// SIMATIC S7-200 project (STEP 7-Micro/WIN), CPU 221 REL 01.10

ORGANIZATION_BLOCK PRINCIPAL:OB1
TITLE=COMENTARIOS DEL PROGRAMA
BEGIN
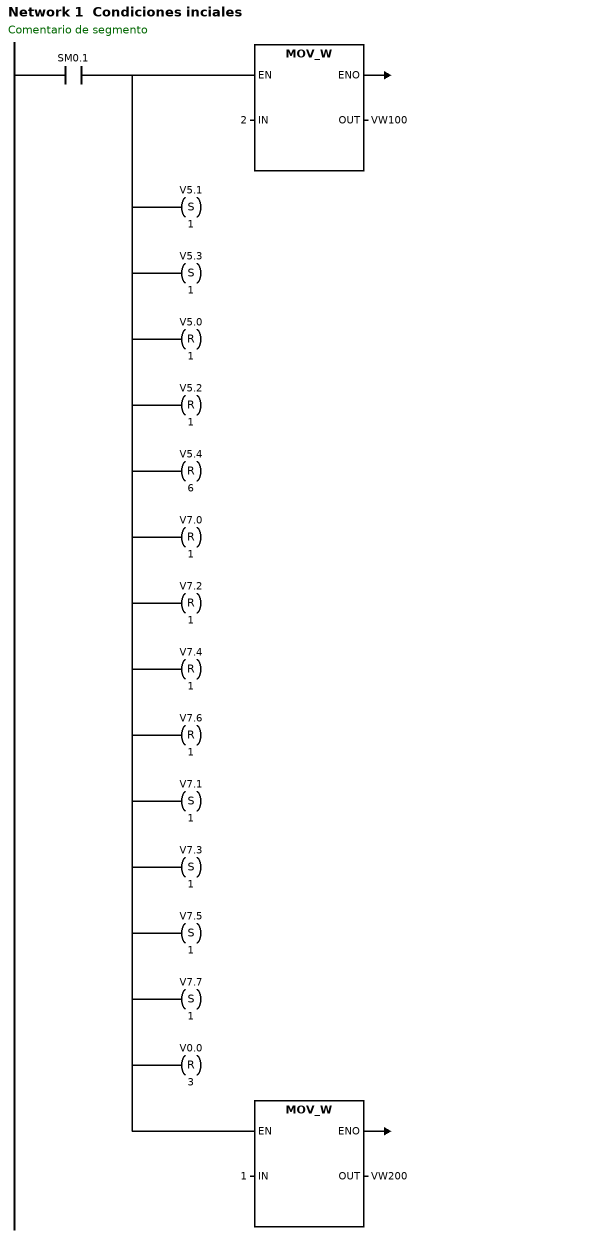
Network 1 // Condiciones inciales
// Comentario de segmento
LD     SM0.1
MOVW   2, VW100
S      V5.1, 1
S      V5.3, 1
R      V5.0, 1
R      V5.2, 1
R      V5.4, 6
R      V7.0, 1
R      V7.2, 1
R      V7.4, 1
R      V7.6, 1
S      V7.1, 1
S      V7.3, 1
S      V7.5, 1
S      V7.7, 1
R      V0.0, 3
MOVW   1, VW200
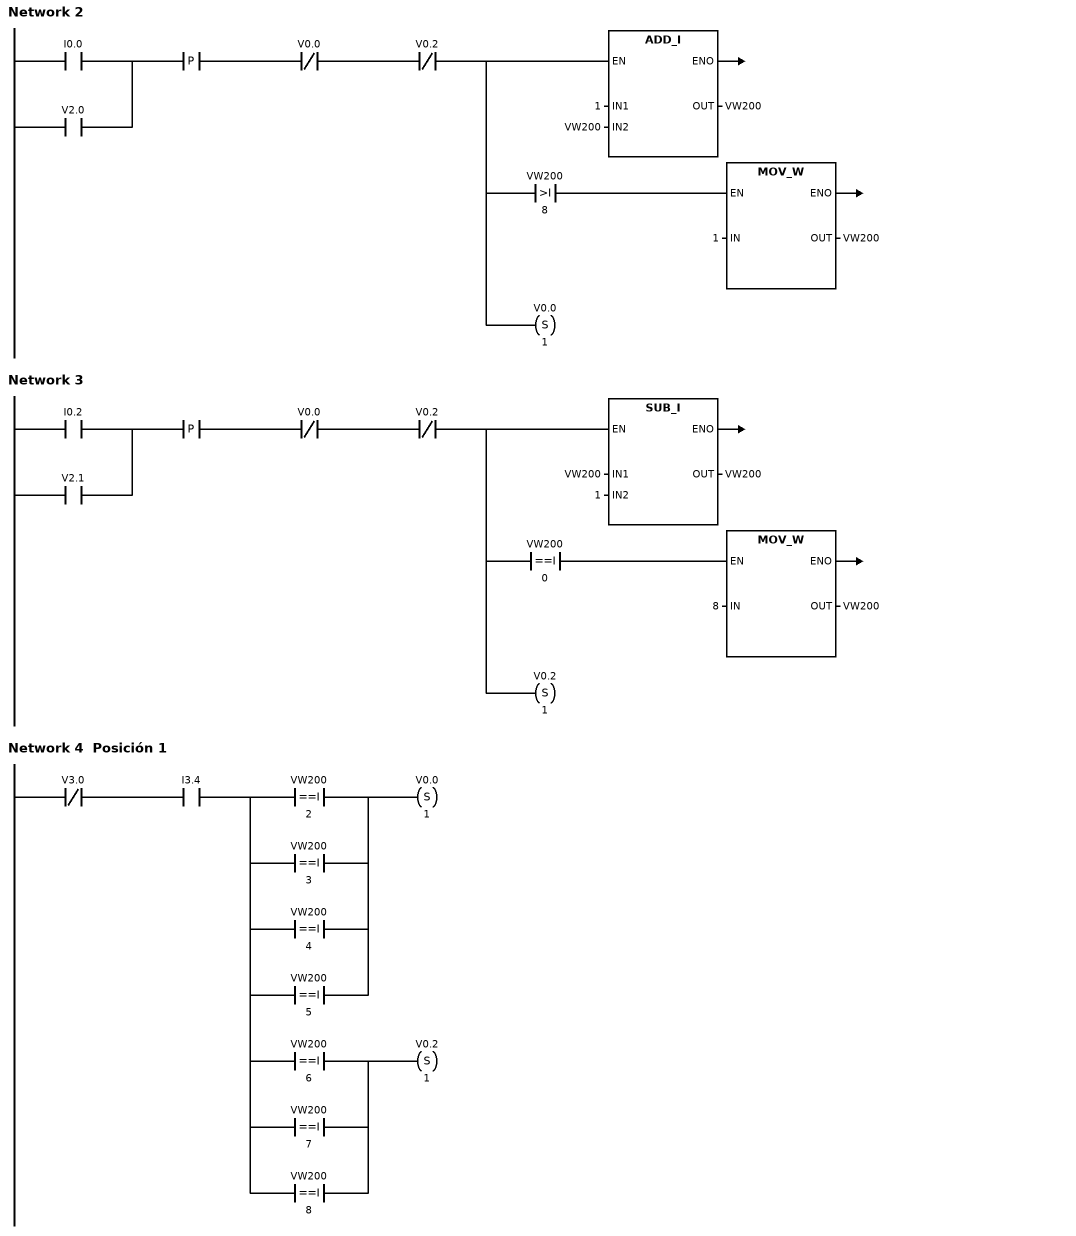
Network 2
LD     I0.0
O      V2.0
EU
AN     V0.0
AN     V0.2
LPS
+I     1, VW200
AW>    VW200, 8
MOVW   1, VW200
LPP
S      V0.0, 1
Network 3
LD     I0.2
O      V2.1
EU
AN     V0.0
AN     V0.2
LPS
-I     1, VW200
AW=    VW200, 0
MOVW   8, VW200
LPP
S      V0.2, 1
Network 4 // Posición 1
LDN    V3.0
A      I3.4
LPS
LDW=   VW200, 2
OW=    VW200, 3
OW=    VW200, 4
OW=    VW200, 5
ALD
S      V0.0, 1
LPP
LDW=   VW200, 6
OW=    VW200, 7
OW=    VW200, 8
ALD
S      V0.2, 1
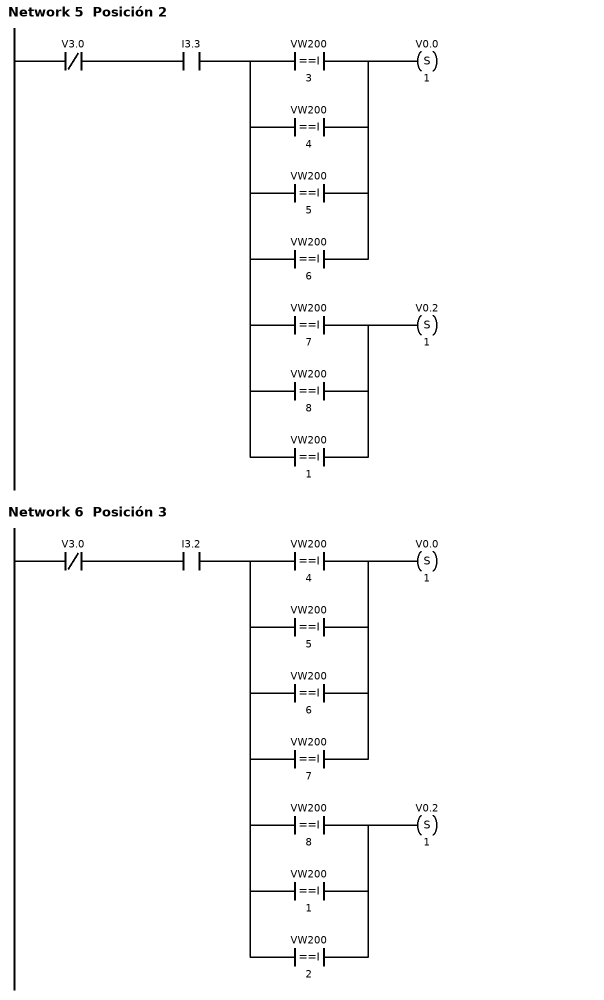
Network 5 // Posición 2
LDN    V3.0
A      I3.3
LPS
LDW=   VW200, 3
OW=    VW200, 4
OW=    VW200, 5
OW=    VW200, 6
ALD
S      V0.0, 1
LPP
LDW=   VW200, 7
OW=    VW200, 8
OW=    VW200, 1
ALD
S      V0.2, 1
Network 6 // Posición 3
LDN    V3.0
A      I3.2
LPS
LDW=   VW200, 4
OW=    VW200, 5
OW=    VW200, 6
OW=    VW200, 7
ALD
S      V0.0, 1
LPP
LDW=   VW200, 8
OW=    VW200, 1
OW=    VW200, 2
ALD
S      V0.2, 1
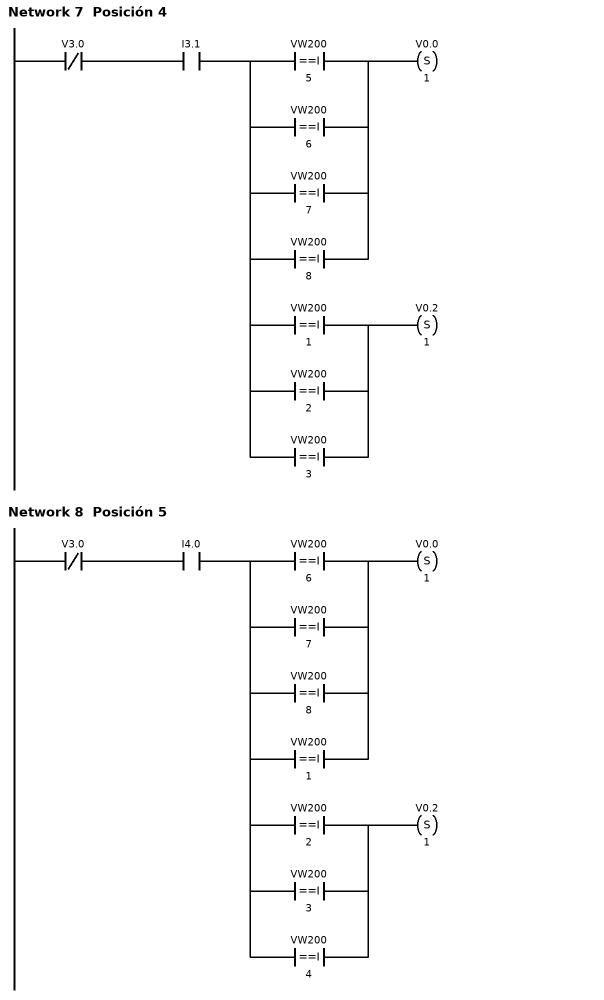
Network 7 // Posición 4
LDN    V3.0
A      I3.1
LPS
LDW=   VW200, 5
OW=    VW200, 6
OW=    VW200, 7
OW=    VW200, 8
ALD
S      V0.0, 1
LPP
LDW=   VW200, 1
OW=    VW200, 2
OW=    VW200, 3
ALD
S      V0.2, 1
Network 8 // Posición 5
LDN    V3.0
A      I4.0
LPS
LDW=   VW200, 6
OW=    VW200, 7
OW=    VW200, 8
OW=    VW200, 1
ALD
S      V0.0, 1
LPP
LDW=   VW200, 2
OW=    VW200, 3
OW=    VW200, 4
ALD
S      V0.2, 1
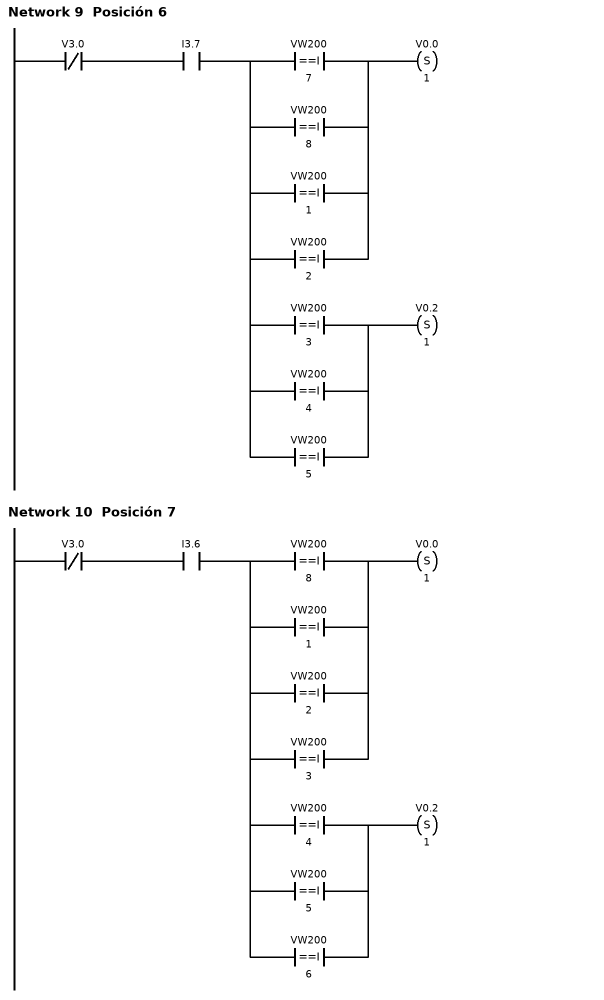
Network 9 // Posición 6
LDN    V3.0
A      I3.7
LPS
LDW=   VW200, 7
OW=    VW200, 8
OW=    VW200, 1
OW=    VW200, 2
ALD
S      V0.0, 1
LPP
LDW=   VW200, 3
OW=    VW200, 4
OW=    VW200, 5
ALD
S      V0.2, 1
Network 10 // Posición 7
LDN    V3.0
A      I3.6
LPS
LDW=   VW200, 8
OW=    VW200, 1
OW=    VW200, 2
OW=    VW200, 3
ALD
S      V0.0, 1
LPP
LDW=   VW200, 4
OW=    VW200, 5
OW=    VW200, 6
ALD
S      V0.2, 1
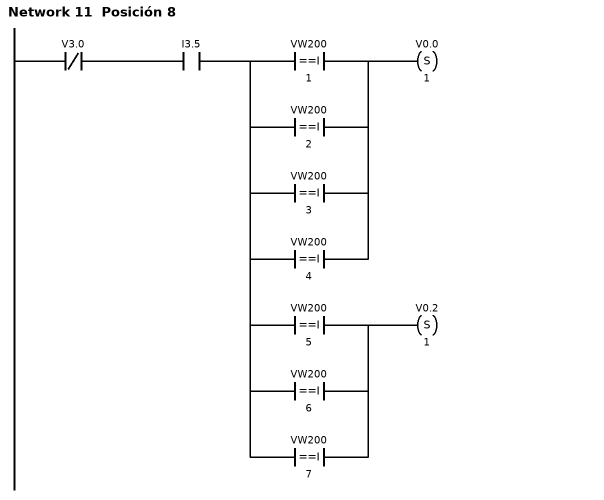
Network 11 // Posición 8
LDN    V3.0
A      I3.5
LPS
LDW=   VW200, 1
OW=    VW200, 2
OW=    VW200, 3
OW=    VW200, 4
ALD
S      V0.0, 1
LPP
LDW=   VW200, 5
OW=    VW200, 6
OW=    VW200, 7
ALD
S      V0.2, 1
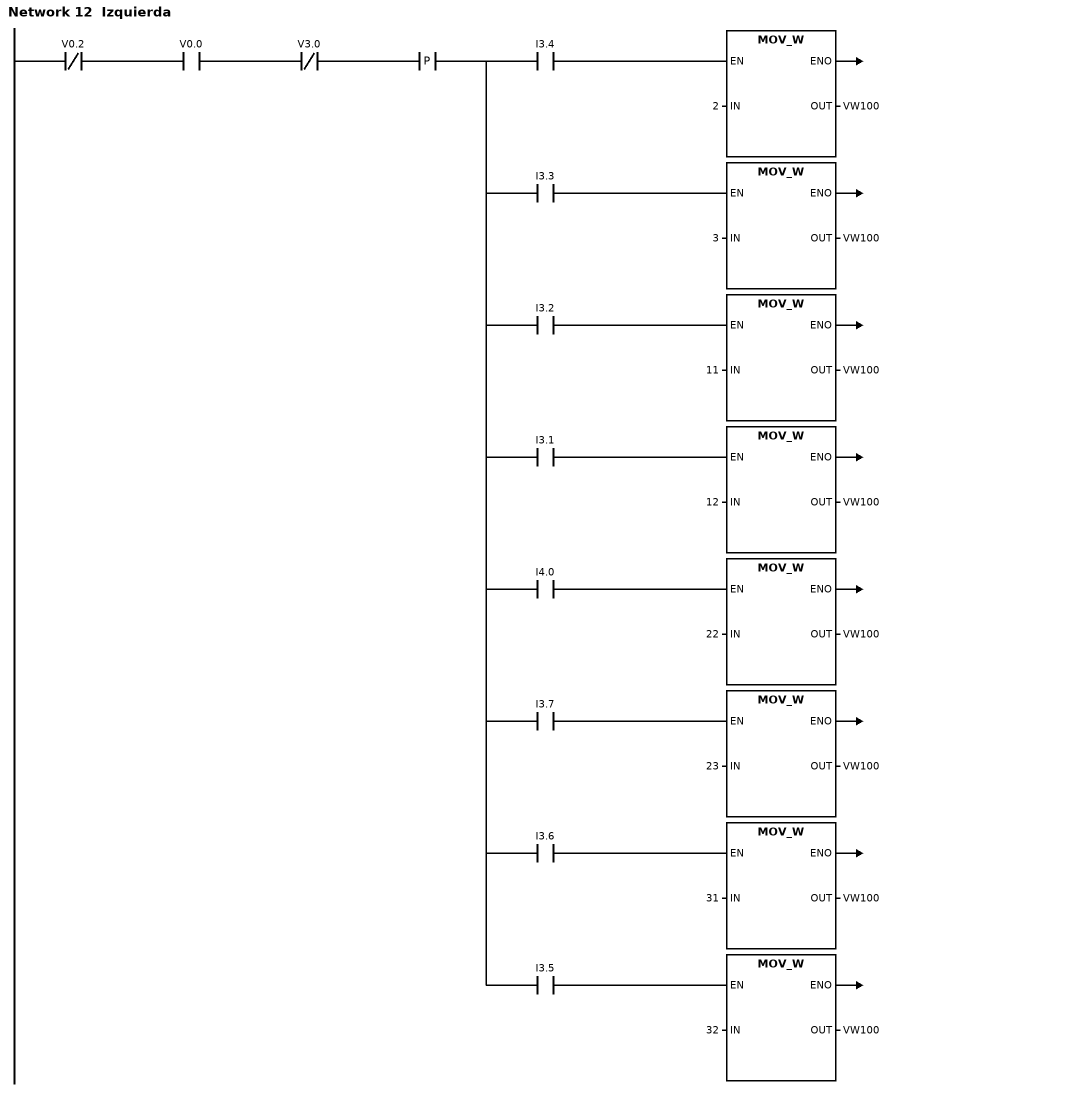
Network 12 // Izquierda
LDN    V0.2
A      V0.0
AN     V3.0
EU
LPS
A      I3.4
MOVW   2, VW100
LRD
A      I3.3
MOVW   3, VW100
LRD
A      I3.2
MOVW   11, VW100
LRD
A      I3.1
MOVW   12, VW100
LRD
A      I4.0
MOVW   22, VW100
LRD
A      I3.7
MOVW   23, VW100
LRD
A      I3.6
MOVW   31, VW100
LPP
A      I3.5
MOVW   32, VW100
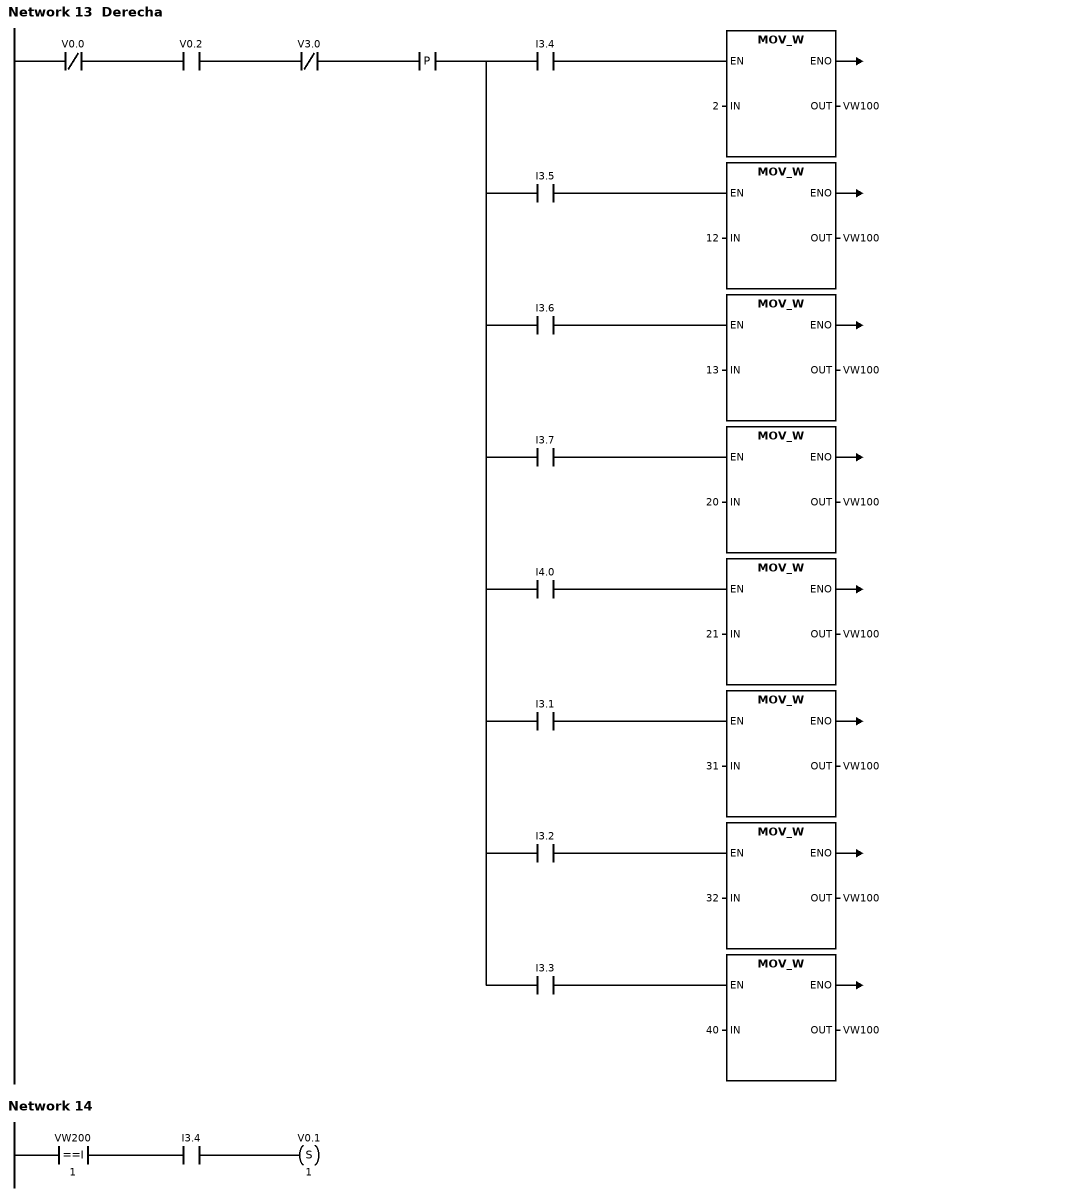
Network 13 // Derecha
LDN    V0.0
A      V0.2
AN     V3.0
EU
LPS
A      I3.4
MOVW   2, VW100
LRD
A      I3.5
MOVW   12, VW100
LRD
A      I3.6
MOVW   13, VW100
LRD
A      I3.7
MOVW   20, VW100
LRD
A      I4.0
MOVW   21, VW100
LRD
A      I3.1
MOVW   31, VW100
LRD
A      I3.2
MOVW   32, VW100
LPP
A      I3.3
MOVW   40, VW100
Network 14
LDW=   VW200, 1
A      I3.4
S      V0.1, 1
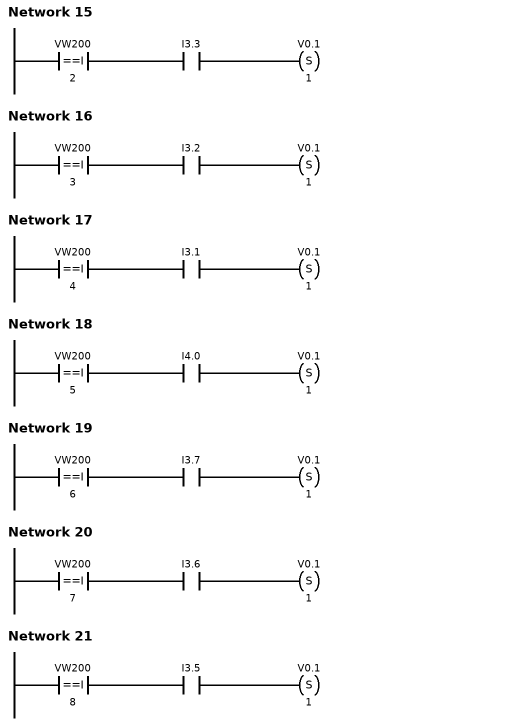
Network 15
LDW=   VW200, 2
A      I3.3
S      V0.1, 1
Network 16
LDW=   VW200, 3
A      I3.2
S      V0.1, 1
Network 17
LDW=   VW200, 4
A      I3.1
S      V0.1, 1
Network 18
LDW=   VW200, 5
A      I4.0
S      V0.1, 1
Network 19
LDW=   VW200, 6
A      I3.7
S      V0.1, 1
Network 20
LDW=   VW200, 7
A      I3.6
S      V0.1, 1
Network 21
LDW=   VW200, 8
A      I3.5
S      V0.1, 1
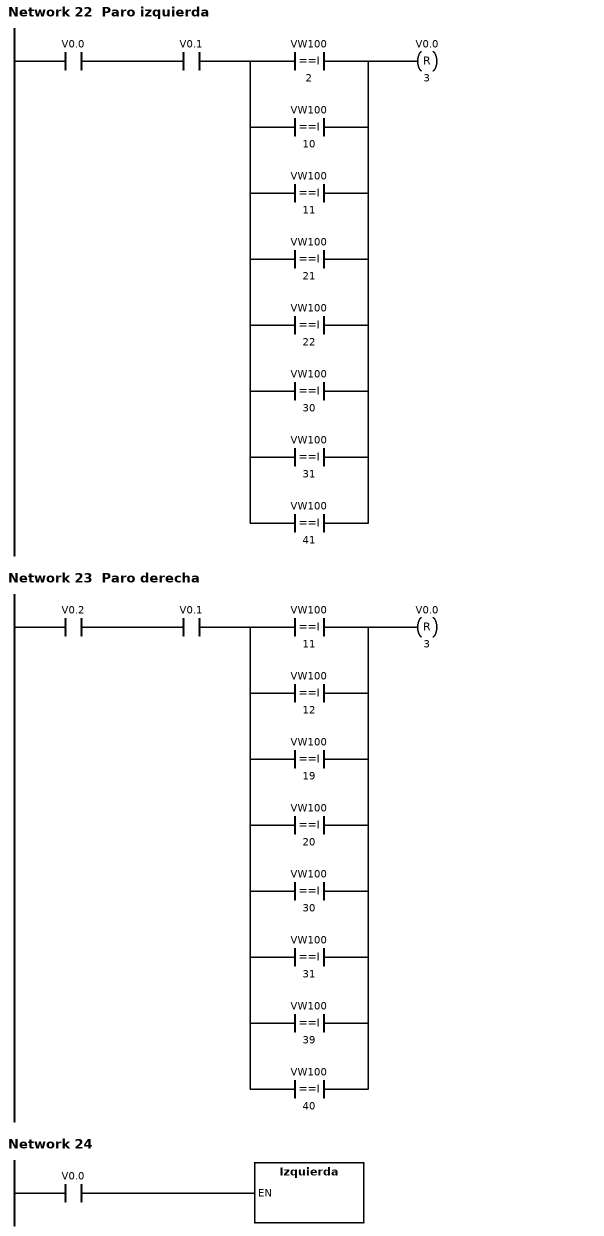
Network 22 // Paro izquierda
LD     V0.0
A      V0.1
LDW=   VW100, 2
OW=    VW100, 10
OW=    VW100, 11
OW=    VW100, 21
OW=    VW100, 22
OW=    VW100, 30
OW=    VW100, 31
OW=    VW100, 41
ALD
R      V0.0, 3
Network 23 // Paro derecha
LD     V0.2
A      V0.1
LDW=   VW100, 11
OW=    VW100, 12
OW=    VW100, 19
OW=    VW100, 20
OW=    VW100, 30
OW=    VW100, 31
OW=    VW100, 39
OW=    VW100, 40
ALD
R      V0.0, 3
Network 24
LD     V0.0
CALL   Izquierda:SBR0
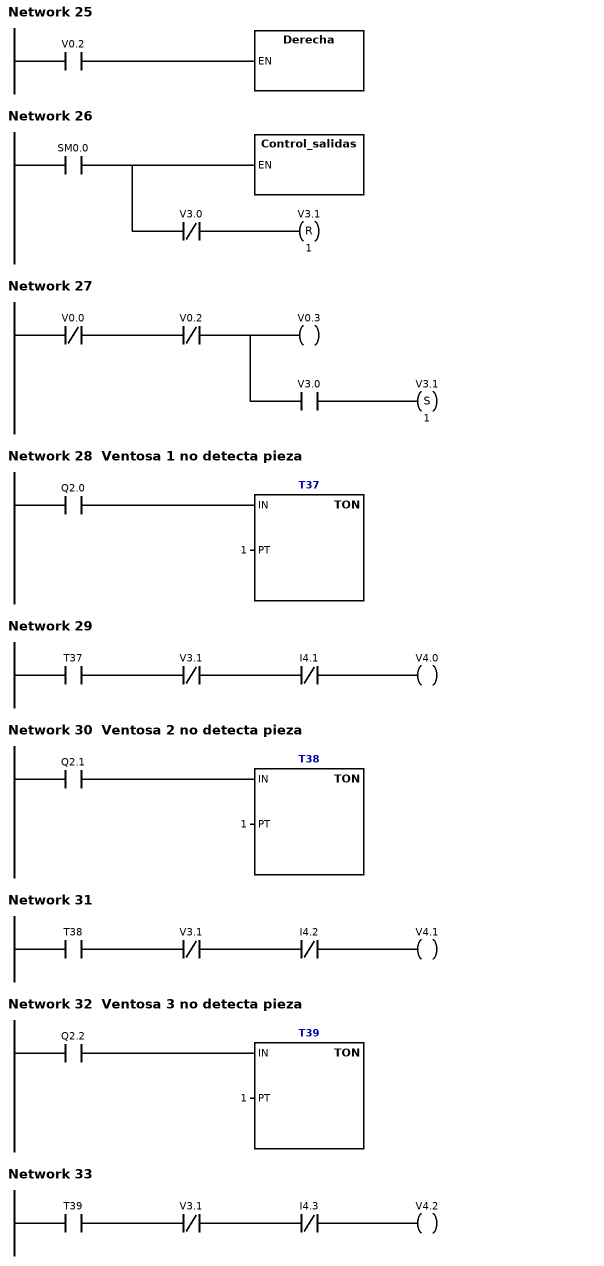
Network 25
LD     V0.2
CALL   Derecha:SBR1
Network 26
LD     SM0.0
CALL   Control_salidas:SBR2
AN     V3.0
R      V3.1, 1
Network 27
LDN    V0.0
AN     V0.2
=      V0.3
A      V3.0
S      V3.1, 1
Network 28 // Ventosa 1 no detecta pieza
LD     Q2.0
TON    T37, 1
Network 29
LD     T37
AN     V3.1
AN     I4.1
=      V4.0
Network 30 // Ventosa 2 no detecta pieza
LD     Q2.1
TON    T38, 1
Network 31
LD     T38
AN     V3.1
AN     I4.2
=      V4.1
Network 32 // Ventosa 3 no detecta pieza
LD     Q2.2
TON    T39, 1
Network 33
LD     T39
AN     V3.1
AN     I4.3
=      V4.2
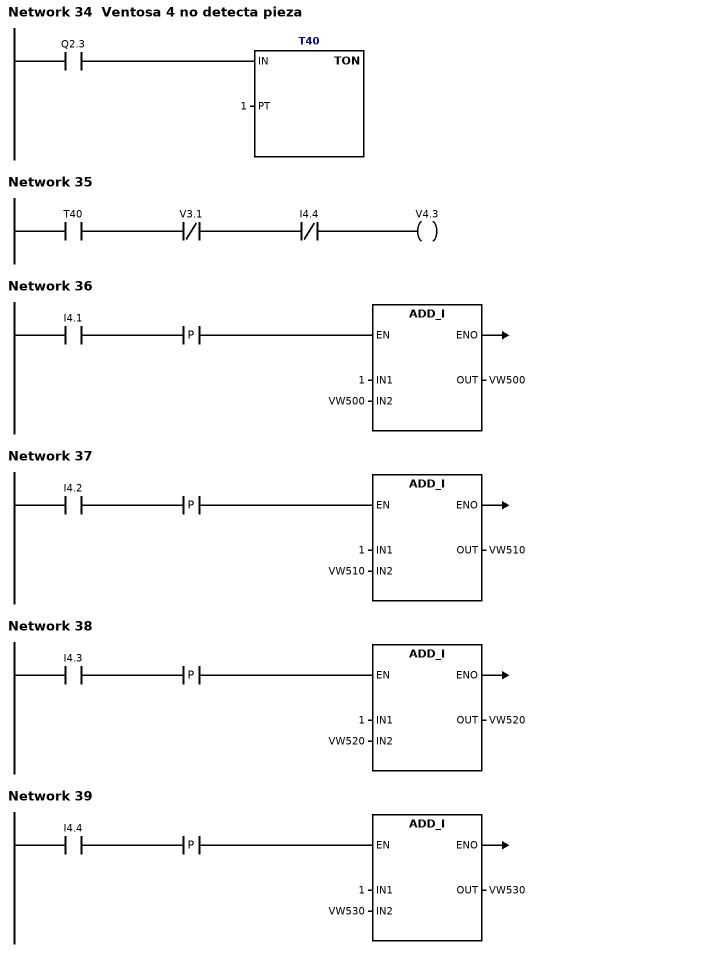
Network 34 // Ventosa 4 no detecta pieza
LD     Q2.3
TON    T40, 1
Network 35
LD     T40
AN     V3.1
AN     I4.4
=      V4.3
Network 36
LD     I4.1
EU
+I     1, VW500
Network 37
LD     I4.2
EU
+I     1, VW510
Network 38
LD     I4.3
EU
+I     1, VW520
Network 39
LD     I4.4
EU
+I     1, VW530
END_ORGANIZATION_BLOCK

SUBROUTINE_BLOCK Izquierda:SBR0
TITLE=COMENTARIOS DE LA SUBRUTINA
BEGIN
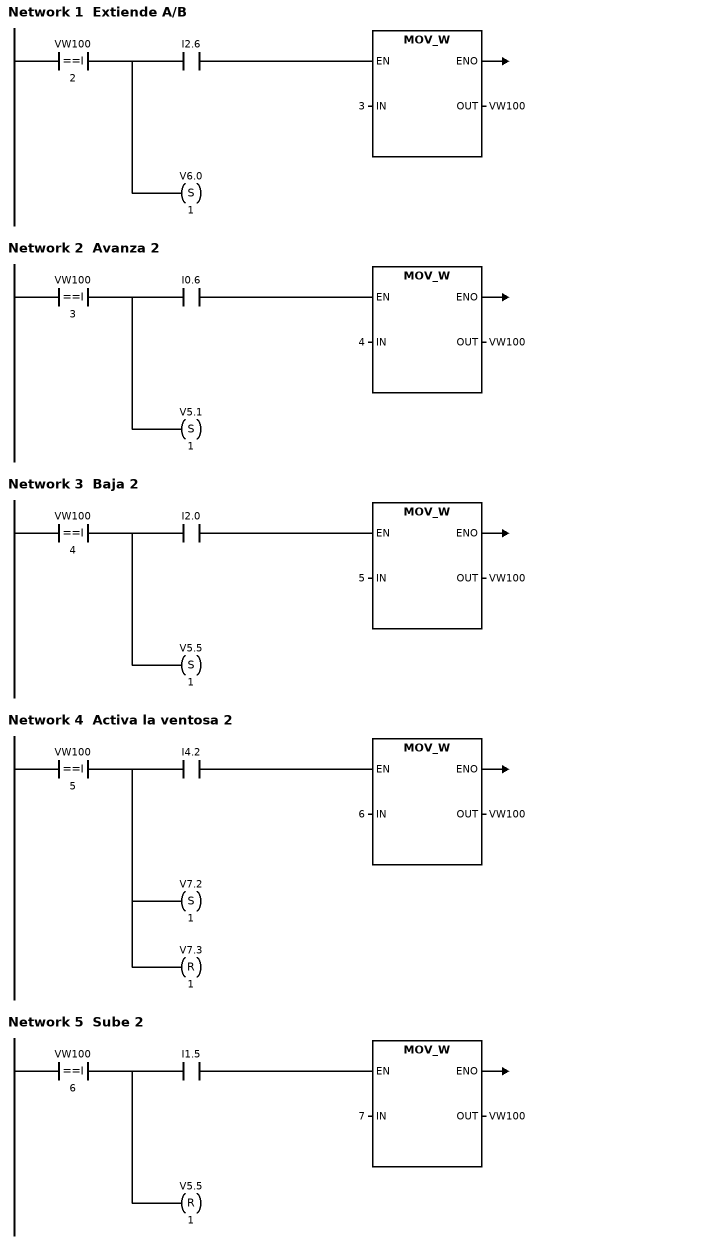
Network 1 // Extiende A/B
LDW=   VW100, 2
LPS
A      I2.6
MOVW   3, VW100
LPP
S      V6.0, 1
Network 2 // Avanza 2
LDW=   VW100, 3
LPS
A      I0.6
MOVW   4, VW100
LPP
S      V5.1, 1
Network 3 // Baja 2
LDW=   VW100, 4
LPS
A      I2.0
MOVW   5, VW100
LPP
S      V5.5, 1
Network 4 // Activa la ventosa 2
LDW=   VW100, 5
LPS
A      I4.2
MOVW   6, VW100
LRD
S      V7.2, 1
LPP
R      V7.3, 1
Network 5 // Sube 2
LDW=   VW100, 6
LPS
A      I1.5
MOVW   7, VW100
LPP
R      V5.5, 1
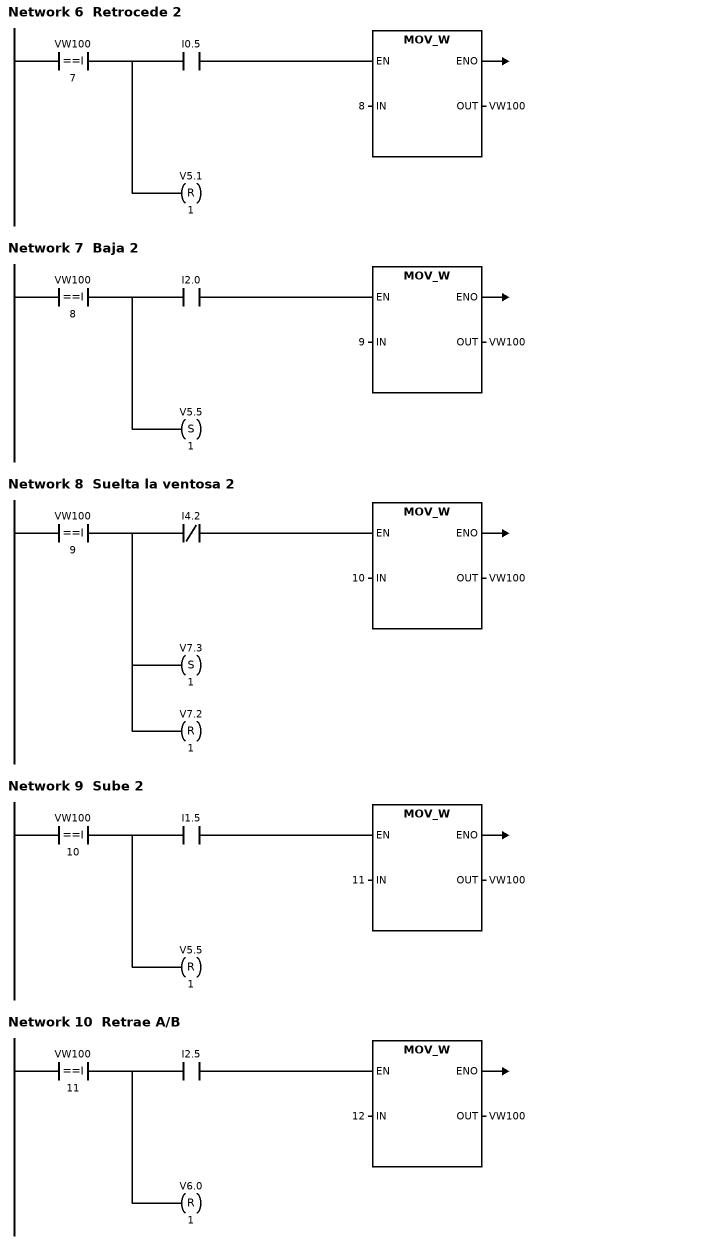
Network 6 // Retrocede 2
LDW=   VW100, 7
LPS
A      I0.5
MOVW   8, VW100
LPP
R      V5.1, 1
Network 7 // Baja 2
LDW=   VW100, 8
LPS
A      I2.0
MOVW   9, VW100
LPP
S      V5.5, 1
Network 8 // Suelta la ventosa 2
LDW=   VW100, 9
LPS
AN     I4.2
MOVW   10, VW100
LRD
S      V7.3, 1
LPP
R      V7.2, 1
Network 9 // Sube 2
LDW=   VW100, 10
LPS
A      I1.5
MOVW   11, VW100
LPP
R      V5.5, 1
Network 10 // Retrae A/B
LDW=   VW100, 11
LPS
A      I2.5
MOVW   12, VW100
LPP
R      V6.0, 1
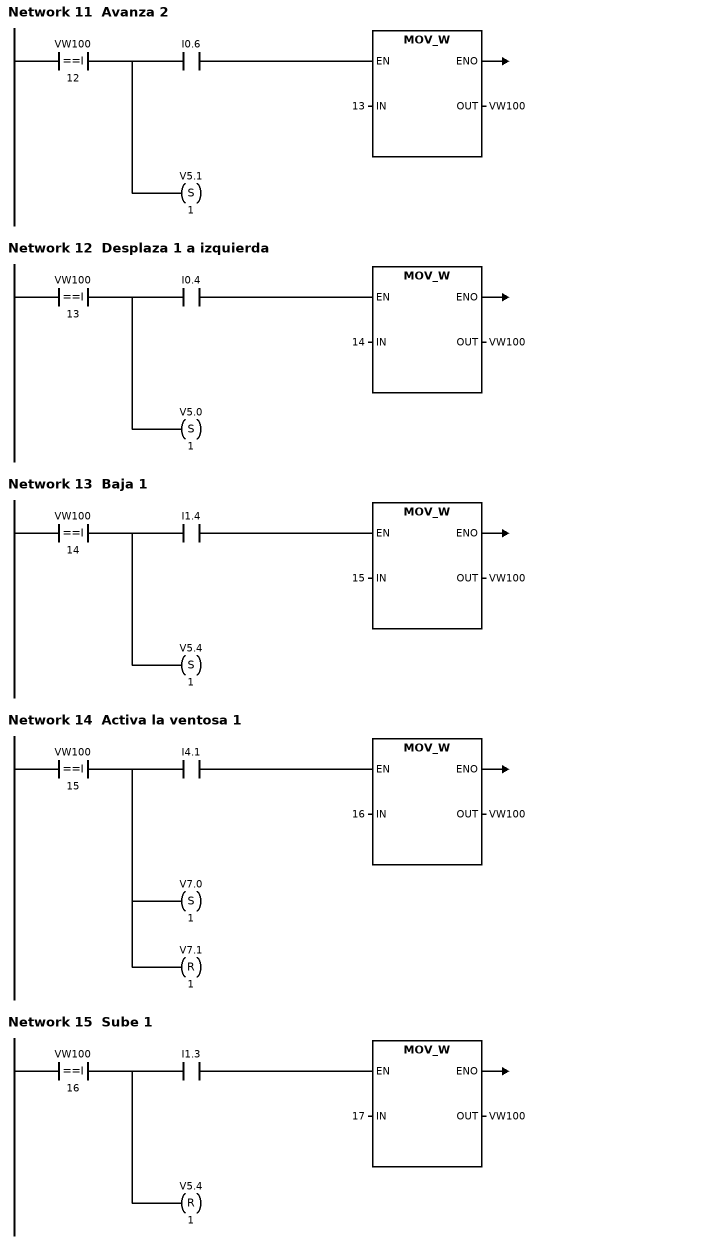
Network 11 // Avanza 2
LDW=   VW100, 12
LPS
A      I0.6
MOVW   13, VW100
LPP
S      V5.1, 1
Network 12 // Desplaza 1 a izquierda
LDW=   VW100, 13
LPS
A      I0.4
MOVW   14, VW100
LPP
S      V5.0, 1
Network 13 // Baja 1
LDW=   VW100, 14
LPS
A      I1.4
MOVW   15, VW100
LPP
S      V5.4, 1
Network 14 // Activa la ventosa 1
LDW=   VW100, 15
LPS
A      I4.1
MOVW   16, VW100
LRD
S      V7.0, 1
LPP
R      V7.1, 1
Network 15 // Sube 1
LDW=   VW100, 16
LPS
A      I1.3
MOVW   17, VW100
LPP
R      V5.4, 1
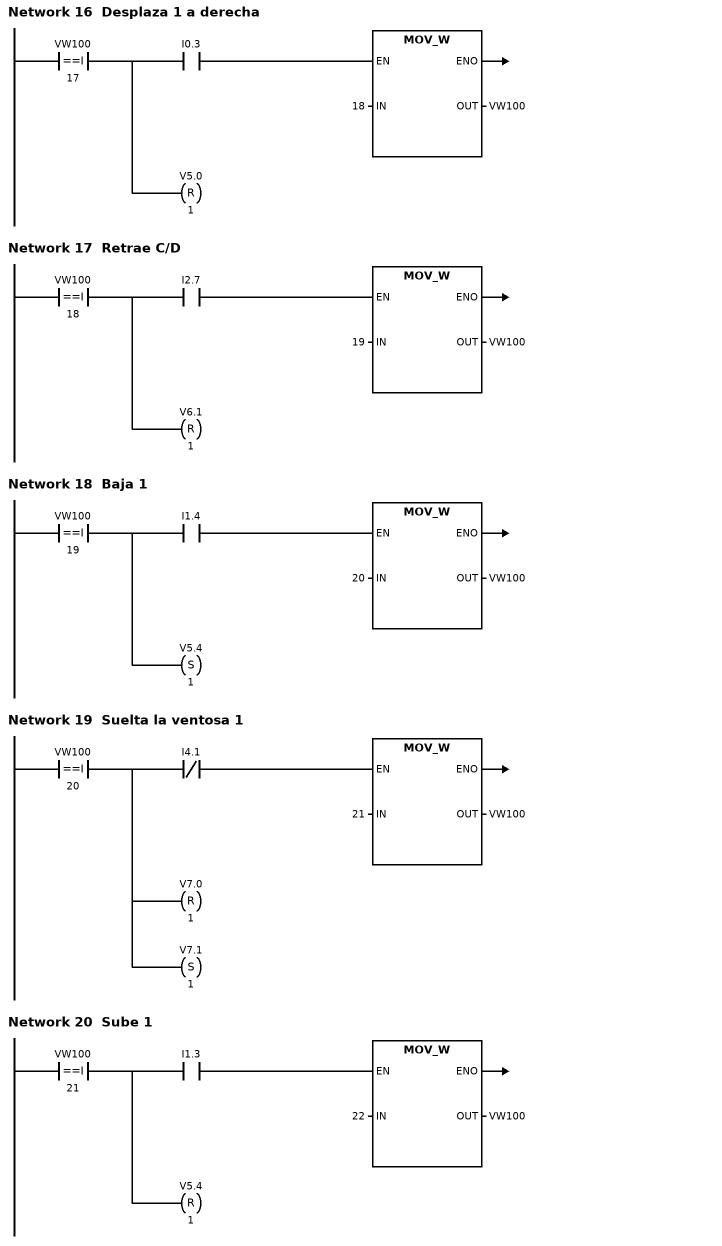
Network 16 // Desplaza 1 a derecha
LDW=   VW100, 17
LPS
A      I0.3
MOVW   18, VW100
LPP
R      V5.0, 1
Network 17 // Retrae C/D
LDW=   VW100, 18
LPS
A      I2.7
MOVW   19, VW100
LPP
R      V6.1, 1
Network 18 // Baja 1
LDW=   VW100, 19
LPS
A      I1.4
MOVW   20, VW100
LPP
S      V5.4, 1
Network 19 // Suelta la ventosa 1
LDW=   VW100, 20
LPS
AN     I4.1
MOVW   21, VW100
LRD
R      V7.0, 1
LPP
S      V7.1, 1
Network 20 // Sube 1
LDW=   VW100, 21
LPS
A      I1.3
MOVW   22, VW100
LPP
R      V5.4, 1
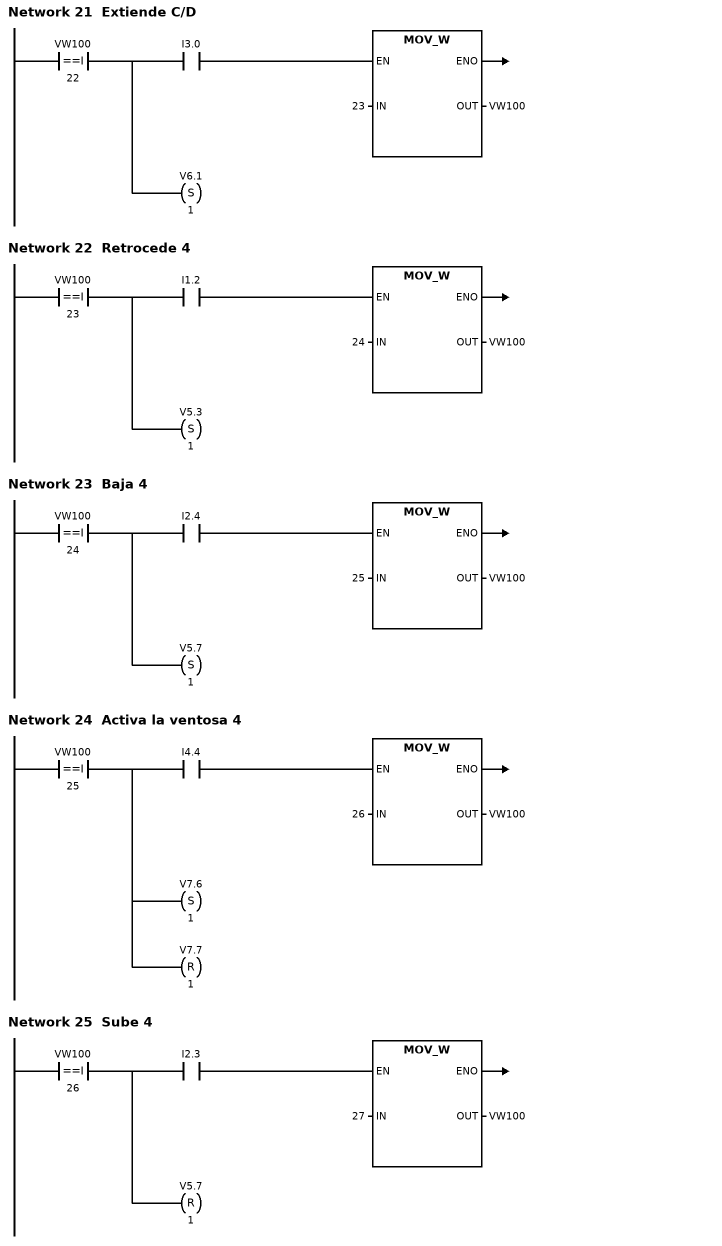
Network 21 // Extiende C/D
LDW=   VW100, 22
LPS
A      I3.0
MOVW   23, VW100
LPP
S      V6.1, 1
Network 22 // Retrocede 4
LDW=   VW100, 23
LPS
A      I1.2
MOVW   24, VW100
LPP
S      V5.3, 1
Network 23 // Baja 4
LDW=   VW100, 24
LPS
A      I2.4
MOVW   25, VW100
LPP
S      V5.7, 1
Network 24 // Activa la ventosa 4
LDW=   VW100, 25
LPS
A      I4.4
MOVW   26, VW100
LRD
S      V7.6, 1
LPP
R      V7.7, 1
Network 25 // Sube 4
LDW=   VW100, 26
LPS
A      I2.3
MOVW   27, VW100
LPP
R      V5.7, 1
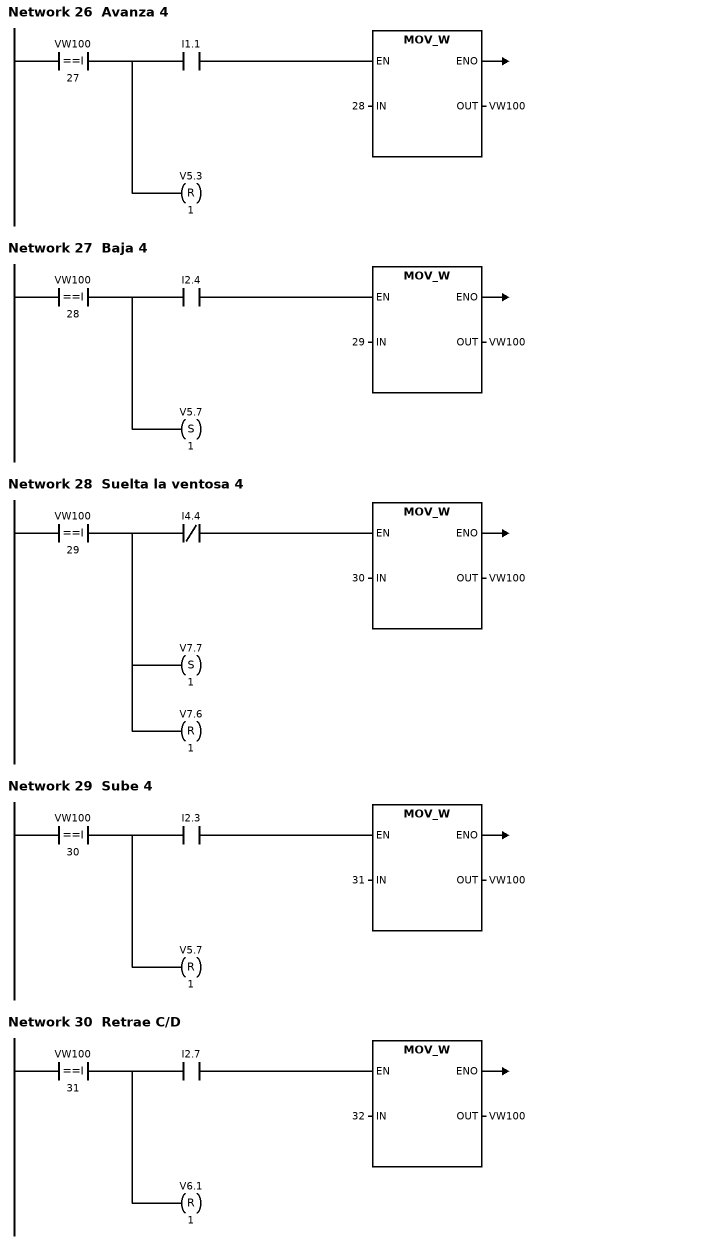
Network 26 // Avanza 4
LDW=   VW100, 27
LPS
A      I1.1
MOVW   28, VW100
LPP
R      V5.3, 1
Network 27 // Baja 4
LDW=   VW100, 28
LPS
A      I2.4
MOVW   29, VW100
LPP
S      V5.7, 1
Network 28 // Suelta la ventosa 4
LDW=   VW100, 29
LPS
AN     I4.4
MOVW   30, VW100
LRD
S      V7.7, 1
LPP
R      V7.6, 1
Network 29 // Sube 4
LDW=   VW100, 30
LPS
A      I2.3
MOVW   31, VW100
LPP
R      V5.7, 1
Network 30 // Retrae C/D
LDW=   VW100, 31
LPS
A      I2.7
MOVW   32, VW100
LPP
R      V6.1, 1
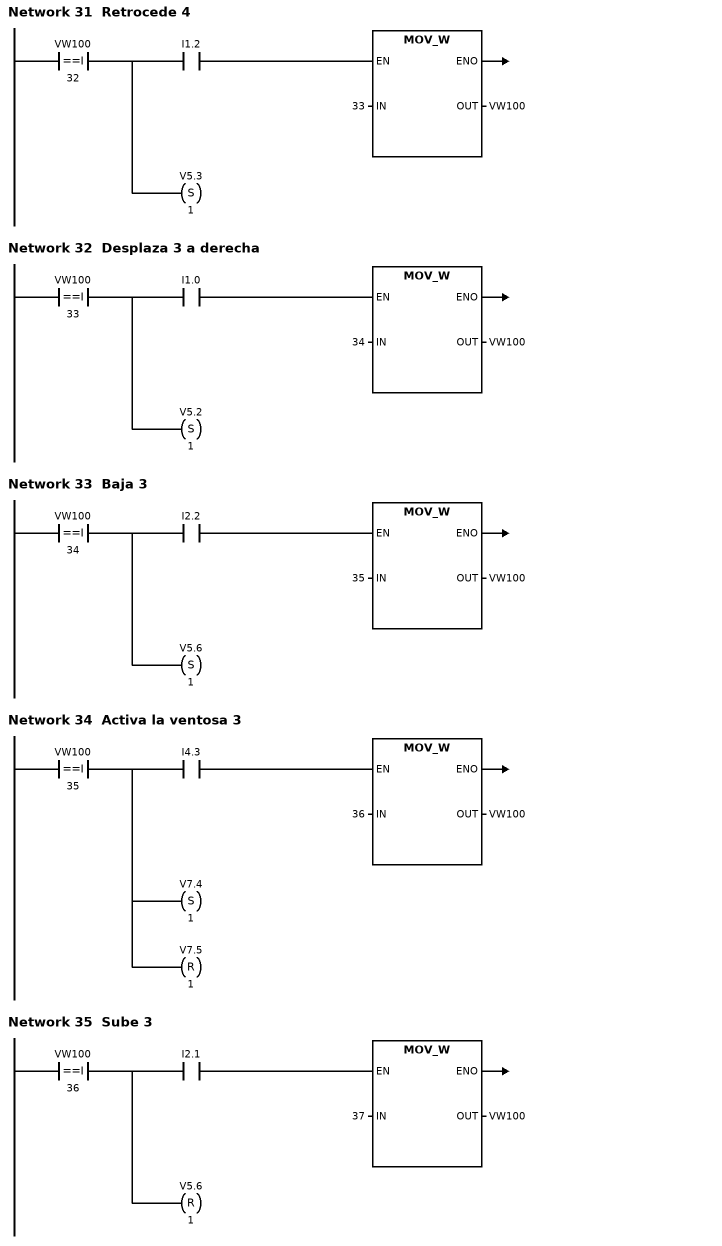
Network 31 // Retrocede 4
LDW=   VW100, 32
LPS
A      I1.2
MOVW   33, VW100
LPP
S      V5.3, 1
Network 32 // Desplaza 3 a derecha
LDW=   VW100, 33
LPS
A      I1.0
MOVW   34, VW100
LPP
S      V5.2, 1
Network 33 // Baja 3
LDW=   VW100, 34
LPS
A      I2.2
MOVW   35, VW100
LPP
S      V5.6, 1
Network 34 // Activa la ventosa 3
LDW=   VW100, 35
LPS
A      I4.3
MOVW   36, VW100
LRD
S      V7.4, 1
LPP
R      V7.5, 1
Network 35 // Sube 3
LDW=   VW100, 36
LPS
A      I2.1
MOVW   37, VW100
LPP
R      V5.6, 1
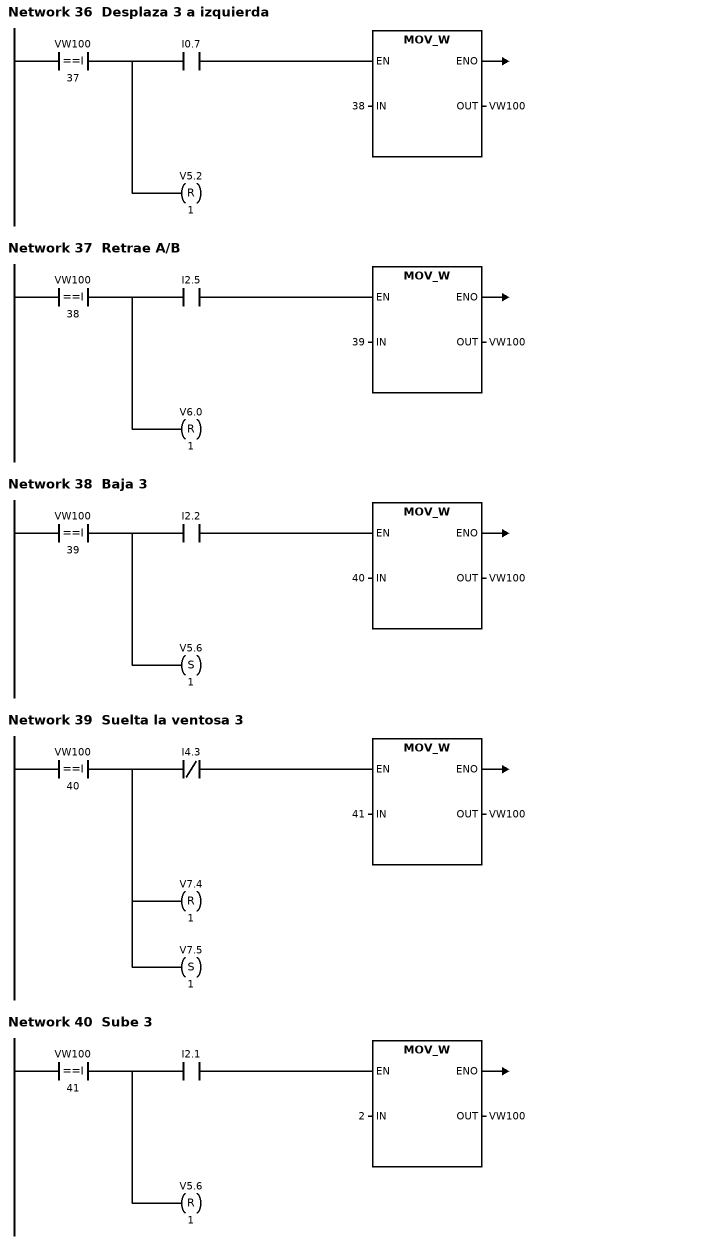
Network 36 // Desplaza 3 a izquierda
LDW=   VW100, 37
LPS
A      I0.7
MOVW   38, VW100
LPP
R      V5.2, 1
Network 37 // Retrae A/B
LDW=   VW100, 38
LPS
A      I2.5
MOVW   39, VW100
LPP
R      V6.0, 1
Network 38 // Baja 3
LDW=   VW100, 39
LPS
A      I2.2
MOVW   40, VW100
LPP
S      V5.6, 1
Network 39 // Suelta la ventosa 3
LDW=   VW100, 40
LPS
AN     I4.3
MOVW   41, VW100
LRD
R      V7.4, 1
LPP
S      V7.5, 1
Network 40 // Sube 3
LDW=   VW100, 41
LPS
A      I2.1
MOVW   2, VW100
LPP
R      V5.6, 1
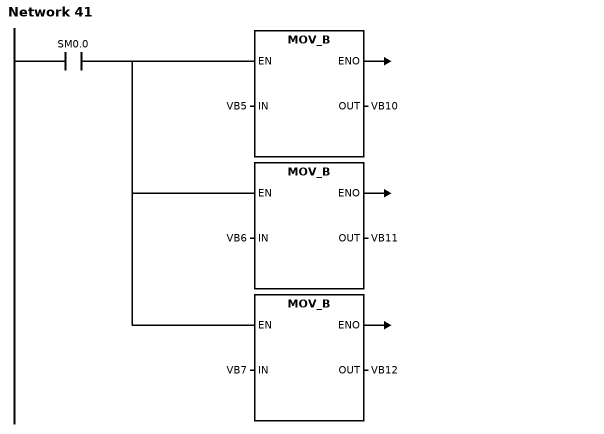
Network 41
LD     SM0.0
MOVB   VB5, VB10
MOVB   VB6, VB11
MOVB   VB7, VB12
END_SUBROUTINE_BLOCK

SUBROUTINE_BLOCK Derecha:SBR1
TITLE=COMENTARIOS DE LA SUBRUTINA
BEGIN
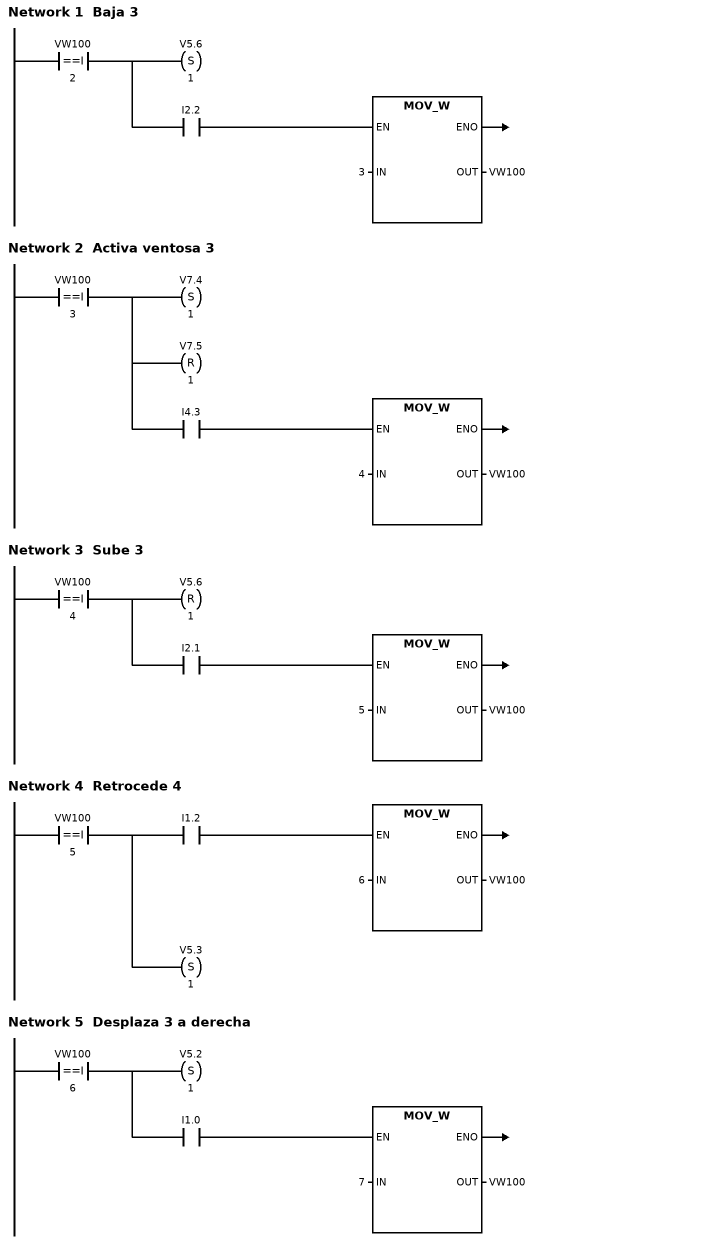
Network 1 // Baja 3
LDW=   VW100, 2
S      V5.6, 1
A      I2.2
MOVW   3, VW100
Network 2 // Activa ventosa 3
LDW=   VW100, 3
S      V7.4, 1
R      V7.5, 1
A      I4.3
MOVW   4, VW100
Network 3 // Sube 3
LDW=   VW100, 4
R      V5.6, 1
A      I2.1
MOVW   5, VW100
Network 4 // Retrocede 4
LDW=   VW100, 5
LPS
A      I1.2
MOVW   6, VW100
LPP
S      V5.3, 1
Network 5 // Desplaza 3 a derecha
LDW=   VW100, 6
S      V5.2, 1
A      I1.0
MOVW   7, VW100
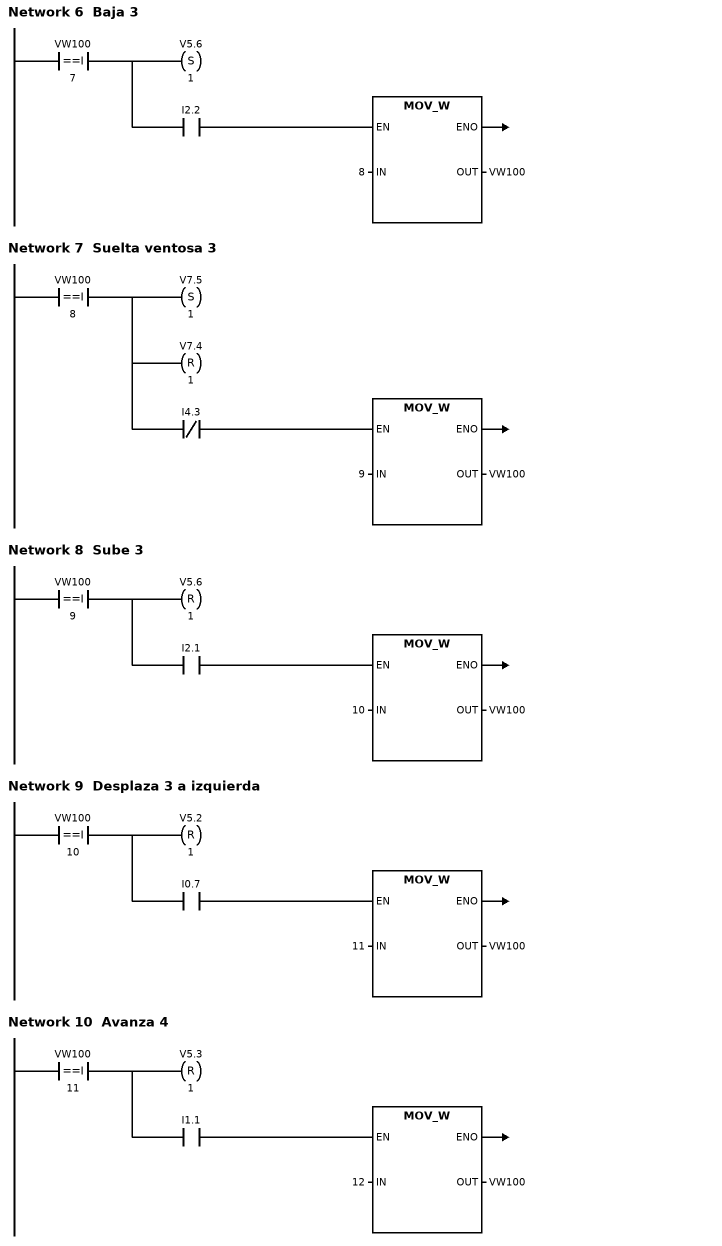
Network 6 // Baja 3
LDW=   VW100, 7
S      V5.6, 1
A      I2.2
MOVW   8, VW100
Network 7 // Suelta ventosa 3
LDW=   VW100, 8
S      V7.5, 1
R      V7.4, 1
AN     I4.3
MOVW   9, VW100
Network 8 // Sube 3
LDW=   VW100, 9
R      V5.6, 1
A      I2.1
MOVW   10, VW100
Network 9 // Desplaza 3 a izquierda
LDW=   VW100, 10
R      V5.2, 1
A      I0.7
MOVW   11, VW100
Network 10 // Avanza 4
LDW=   VW100, 11
R      V5.3, 1
A      I1.1
MOVW   12, VW100
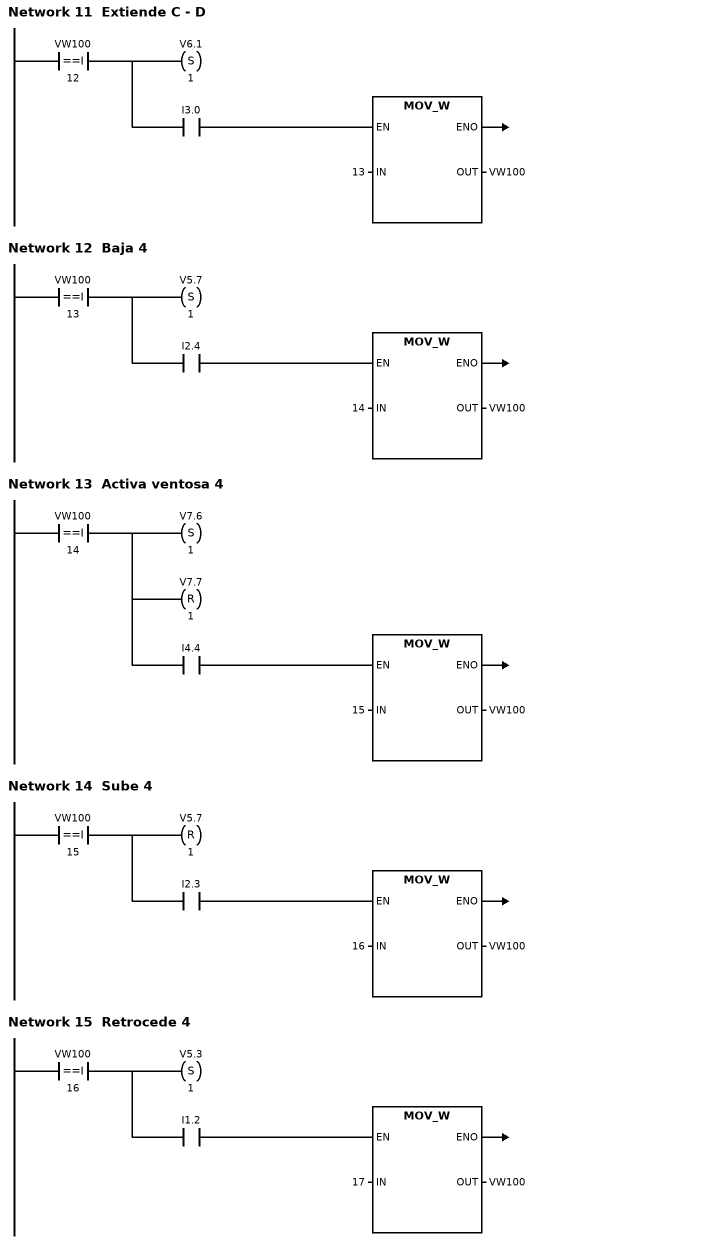
Network 11 // Extiende C - D
LDW=   VW100, 12
S      V6.1, 1
A      I3.0
MOVW   13, VW100
Network 12 // Baja 4
LDW=   VW100, 13
S      V5.7, 1
A      I2.4
MOVW   14, VW100
Network 13 // Activa ventosa 4
LDW=   VW100, 14
S      V7.6, 1
R      V7.7, 1
A      I4.4
MOVW   15, VW100
Network 14 // Sube 4
LDW=   VW100, 15
R      V5.7, 1
A      I2.3
MOVW   16, VW100
Network 15 // Retrocede 4
LDW=   VW100, 16
S      V5.3, 1
A      I1.2
MOVW   17, VW100
